# EPICS autosave request: urRobotApp/Db/path_waypoint_settings.req
$(P)Path$(N):$(K):Type.VAL
$(P)Path$(N):$(K):Number.VAL
$(P)Path$(N):$(K):ActionOverride.VAL
$(P)Path$(N):$(K):Enabled
